{attribute 'reflection'} 
{attribute 'no_explicit_call' := 'do not call this POU directly'} 
FUNCTION_BLOCK FB_STOP_GATE IMPLEMENTS I_STOP_GATE
VAR_INPUT
END_VAR
VAR_OUTPUT
END_VAR
VAR
	{attribute 'instance-path'} 
    {attribute 'noinit'} 
	strInstancePath: STRING;
	strFullObjectPath: STRING;
	stEvent: ST_EVENT;
	bAck: BOOL;
	itfOpMode:				I_OP_MODE;
	itfValveOpenStopGate:	I_BASE_VALVE;
	itfSensorByStopGate: 	I_BINARY_SWITCH;
	itfSensorCongestion: 	I_BINARY_SWITCH;
	
	tonToBase: Tc2_Standard.TON;
	tToBase: TIME;
	tonToWork: Tc2_Standard.TON;
	tToWork: TIME;
	bViewToBase: BOOL;
	bViewToWork: BOOL;
	
	
END_VAR

METHOD FB_init : BOOL
VAR_INPUT
	bInitRetains : BOOL; // if TRUE, the retain variables are initialized (warm start / cold start)
	bInCopyCode : BOOL;  // if TRUE, the instance afterwards gets moved into the copy code (online change)
END_VAR
END_METHOD

{warning 'Methodenimplementierung hinzufügen'}
METHOD M_Close
END_METHOD

{warning 'Methodenimplementierung hinzufügen'}
METHOD M_Open
END_METHOD

{warning 'Methodenimplementierung hinzufügen'}
(*=== Method: M_Run  ============================================

 @brief: Here is the global code (Timer, Event, Flange,...)*)
METHOD M_Run
END_METHOD

{warning 'Methodenimplementierung hinzufügen'}
METHOD M_Seperate
VAR_INPUT
	iCntCarrier	: INT;
END_VAR
END_METHOD


PROPERTY P_CarrierByStopGate : BOOL
GET
END_GET
END_PROPERTY


PROPERTY P_Congestion : BOOL
GET
END_GET
END_PROPERTY


(*=== Property: P_Event  ============================================

 @param [set]: 	Set the Structure "ST_EVENT" from another Object
 @param [get]: 	Return the Structure "ST_EVENT", it contains the actual 
					event of the Object *)
PROPERTY P_Event : ST_EVENT
GET
END_GET
SET
END_SET
END_PROPERTY


(*=== Property: P_FullObjectPath  ============================================

 @param [set]: 	Set the Object Path (Clear String of Object)
 @param [get]: 	Return the Objectpath *)
PROPERTY P_FullObjectPath : STRING
GET
END_GET
SET
END_SET
END_PROPERTY


(*=== Property: P_Global_Ack  ============================================

 @param [set]: 	Set the Bit for Ack from another Object
 @param [get]: 	Return the state of Ack Bit*)
PROPERTY P_Global_Ack : BOOL
GET
END_GET
SET
END_SET
END_PROPERTY


(*=== Property: P_GlobalID  ============================================

 @param [set]: 	-
 @param [get]: 	Return the string of instance path*)
PROPERTY P_GlobalID : STRING
GET
END_GET
END_PROPERTY

END_FUNCTION_BLOCK

(* stored: Version 1.1.0.1, ProductVersion 3.1.4024.12
   POU FB_STOP_GATE: Id {6c87846b-0d5e-4e25-aa10-1fd8ba04cd60}, SpecialFunc None
   Method FB_init: Id {9f238b89-a8eb-46d7-bade-6edcb946518f}
   Method M_Close: Id {f095a0e5-08dd-4684-8d1c-fdc58c1a1dc9}
   Method M_Open: Id {ebfb7bcf-289f-464c-9ad7-d2d176ed6185}
   Method M_Run: Id {8a855a35-0833-4a9f-b28b-df3703f5fc08}
   Method M_Seperate: Id {850f7e3b-f59f-42d8-8819-d765e855d36c}
   Property P_CarrierByStopGate: Id {12c045a0-37e2-4fc6-b295-b354b256d416}
   Get Get: Id {636615a9-835c-4e54-afb4-da33e93c18ec}
   Property P_Congestion: Id {5c9d1971-bb29-4ab7-b74b-67da4c761ca2}
   Get Get: Id {49c81655-1825-43e4-887c-4e16e2d01db1}
   Property P_Event: Id {56ff248b-14ab-4b88-bdb6-19da5ba6ca6b}
   Get Get: Id {4cb80f78-8228-4ac5-9fc9-e3f089be378c}
   Set Set: Id {035289c2-1f89-40b7-a2a7-929b15678703}
   Property P_FullObjectPath: Id {f56c6fc3-cc94-4614-8e3c-fe067d613b78}
   Get Get: Id {f486a656-b7e4-4525-bfeb-a4e43f627c94}
   Set Set: Id {0858d306-68a1-476a-a472-dc50ab23ea4f}
   Property P_Global_Ack: Id {efa49c73-5214-40a8-b58c-ba55eeb009b0}
   Get Get: Id {7cca04fc-de1a-4ff9-aee3-7d1bb32f222a}
   Set Set: Id {40404ff5-97ae-49fa-a21e-54846416180a}
   Property P_GlobalID: Id {f7d8e9c8-6366-40ae-9bc0-aeca1eeb27f1}
   Get Get: Id {91de927d-ffb9-4641-8c52-fe06e0a5ad71} *)
